MOVL C09799 V=800.0 PL=0
MOVL C09800 V=800.0 PL=0
MOVL C09801 V=800.0 PL=0
MOVL C09802 V=800.0 PL=0
MOVL C09803 V=800.0 PL=0
MOVL C09804 V=800.0 PL=0
MOVL C09805 V=800.0 PL=0
MOVL C09806 V=800.0 PL=0
MOVL C09807 V=800.0 PL=0
MOVL C09808 V=800.0 PL=0
MOVL C09809 V=800.0 PL=0
MOVL C09810 V=800.0 PL=0
MOVL C09811 V=800.0 PL=0
MOVL C09812 V=800.0 PL=0
MOVL C09813 V=800.0 PL=0
MOVL C09814 V=800.0 PL=0
MOVL C09815 V=800.0 PL=0
MOVL C09816 V=800.0 PL=0
MOVL C09817 V=800.0 PL=0
MOVL C09818 V=800.0 PL=0
MOVL C09819 V=800.0 PL=0
MOVL C09820 V=800.0 PL=0
MOVL C09821 V=800.0 PL=0
MOVL C09822 V=800.0 PL=0
MOVL C09823 V=800.0 PL=0
MOVL C09824 V=800.0 PL=0
MOVL C09825 V=800.0 PL=0
MOVL C09826 V=800.0 PL=0
MOVL C09827 V=800.0 PL=0
MOVL C09828 V=800.0 PL=0
MOVL C09829 V=800.0 PL=0
MOVL C09830 V=800.0 PL=0
MOVL C09831 V=800.0 PL=0
MOVL C09832 V=800.0 PL=0
MOVL C09833 V=800.0 PL=0
MOVL C09834 V=800.0 PL=0
MOVL C09835 V=800.0 PL=0
MOVL C09836 V=800.0 PL=0
MOVL C09837 V=800.0 PL=0
MOVL C09838 V=800.0 PL=0
MOVL C09839 V=800.0 PL=0
MOVL C09840 V=800.0 PL=0
MOVL C09841 V=800.0 PL=0
MOVL C09842 V=800.0 PL=0
MOVL C09843 V=800.0 PL=0
MOVL C09844 V=800.0 PL=0
MOVL C09845 V=800.0 PL=0
MOVL C09846 V=800.0 PL=0
MOVL C09847 V=800.0 PL=0
MOVL C09848 V=800.0 PL=0
MOVL C09849 V=800.0 PL=0
MOVL C09850 V=800.0 PL=0
MOVL C09851 V=800.0 PL=0
MOVL C09852 V=800.0 PL=0
MOVL C09853 V=800.0 PL=0
MOVL C09854 V=800.0 PL=0
MOVL C09855 V=800.0 PL=0
MOVL C09856 V=800.0 PL=0
MOVL C09857 V=800.0 PL=0
MOVL C09858 V=800.0 PL=0
MOVL C09859 V=800.0 PL=0
MOVL C09860 V=800.0 PL=0
MOVL C09861 V=800.0 PL=0
MOVL C09862 V=800.0 PL=0
MOVL C09863 V=800.0 PL=0
MOVL C09864 V=800.0 PL=0
MOVL C09865 V=800.0 PL=0
MOVL C09866 V=800.0 PL=0
MOVL C09867 V=800.0 PL=0
MOVL C09868 V=800.0 PL=0
MOVL C09869 V=800.0 PL=0
MOVL C09870 V=800.0 PL=0
MOVL C09871 V=800.0 PL=0
MOVL C09872 V=800.0 PL=0
MOVL C09873 V=800.0 PL=0
MOVL C09874 V=800.0 PL=0
MOVL C09875 V=800.0 PL=0
MOVL C09876 V=800.0 PL=0
MOVL C09877 V=800.0 PL=0
MOVL C09878 V=800.0 PL=0
MOVL C09879 V=800.0 PL=0
MOVL C09880 V=800.0 PL=0
MOVL C09881 V=800.0 PL=0
MOVL C09882 V=800.0 PL=0
MOVL C09883 V=800.0 PL=0
MOVL C09884 V=800.0 PL=0
MOVL C09885 V=800.0 PL=0
MOVL C09886 V=800.0 PL=0
MOVL C09887 V=800.0 PL=0
MOVL C09888 V=800.0 PL=0
MOVL C09889 V=800.0 PL=0
MOVL C09890 V=800.0 PL=0
MOVL C09891 V=800.0 PL=0
MOVL C09892 V=800.0 PL=0
MOVL C09893 V=800.0 PL=0
MOVL C09894 V=800.0 PL=0
MOVL C09895 V=800.0 PL=0
MOVL C09896 V=800.0 PL=0
MOVL C09897 V=800.0 PL=0
MOVL C09898 V=800.0 PL=0
MOVL C09899 V=800.0 PL=0
MOVL C09900 V=800.0 PL=0
MOVL C09901 V=800.0 PL=0
MOVL C09902 V=800.0 PL=0
MOVL C09903 V=800.0 PL=0
MOVL C09904 V=800.0 PL=0
MOVL C09905 V=800.0 PL=0
MOVL C09906 V=800.0 PL=0
MOVL C09907 V=800.0 PL=0
MOVL C09908 V=800.0 PL=0
MOVL C09909 V=800.0 PL=0
MOVL C09910 V=800.0 PL=0
MOVL C09911 V=800.0 PL=0
MOVL C09912 V=800.0 PL=0
MOVL C09913 V=800.0 PL=0
MOVL C09914 V=800.0 PL=0
MOVL C09915 V=800.0 PL=0
MOVL C09916 V=800.0 PL=0
MOVL C09917 V=800.0 PL=0
MOVL C09918 V=800.0 PL=0
MOVL C09919 V=800.0 PL=0
MOVL C09920 V=800.0 PL=0
MOVL C09921 V=800.0 PL=0
MOVL C09922 V=800.0 PL=0
MOVL C09923 V=800.0 PL=0
MOVL C09924 V=800.0 PL=0
MOVL C09925 V=800.0 PL=0
MOVL C09926 V=800.0 PL=0
MOVL C09927 V=800.0 PL=0
MOVL C09928 V=800.0 PL=0
MOVL C09929 V=800.0 PL=0
MOVL C09930 V=800.0 PL=0
MOVL C09931 V=800.0 PL=0
MOVL C09932 V=800.0 PL=0
MOVL C09933 V=800.0 PL=0
MOVL C09934 V=800.0 PL=0
MOVL C09935 V=800.0 PL=0
MOVL C09936 V=800.0 PL=0
MOVL C09937 V=800.0 PL=0
MOVL C09938 V=800.0 PL=0
MOVL C09939 V=800.0 PL=0
MOVL C09940 V=800.0 PL=0
MOVL C09941 V=800.0 PL=0
MOVL C09942 V=800.0 PL=0
MOVL C09943 V=800.0 PL=0
MOVL C09944 V=800.0 PL=0
MOVL C09945 V=800.0 PL=0
MOVL C09946 V=800.0 PL=0
MOVL C09947 V=800.0 PL=0
MOVL C09948 V=800.0 PL=0
MOVL C09949 V=800.0 PL=0
MOVL C09950 V=800.0 PL=0
MOVL C09951 V=800.0 PL=0
MOVL C09952 V=800.0 PL=0
MOVL C09953 V=800.0 PL=0
MOVL C09954 V=800.0 PL=0
MOVL C09955 V=800.0 PL=0
MOVL C09956 V=800.0 PL=0
MOVL C09957 V=800.0 PL=0
MOVL C09958 V=800.0 PL=0
MOVL C09959 V=800.0 PL=0
MOVL C09960 V=800.0 PL=0
MOVL C09961 V=800.0 PL=0
MOVL C09962 V=800.0 PL=0
MOVL C09963 V=800.0 PL=0
MOVL C09964 V=800.0 PL=0
MOVL C09965 V=800.0 PL=0
MOVL C09966 V=800.0 PL=0
MOVL C09967 V=800.0 PL=0
MOVL C09968 V=800.0 PL=0
MOVL C09969 V=800.0 PL=0
MOVL C09970 V=800.0 PL=0
MOVL C09971 V=800.0 PL=0
MOVL C09972 V=800.0 PL=0
MOVL C09973 V=800.0 PL=0
MOVL C09974 V=800.0 PL=0
MOVL C09975 V=800.0 PL=0
MOVL C09976 V=800.0 PL=0
MOVL C09977 V=800.0 PL=0
MOVL C09978 V=800.0 PL=0
MOVL C09979 V=800.0 PL=0
MOVL C09980 V=800.0 PL=0
MOVL C09981 V=800.0 PL=0
MOVL C09982 V=800.0 PL=0
MOVL C09983 V=800.0 PL=0
MOVL C09984 V=800.0 PL=0
MOVL C09985 V=800.0 PL=0
MOVL C09986 V=800.0 PL=0
MOVL C09987 V=800.0 PL=0
MOVL C09988 V=800.0 PL=0
MOVL C09989 V=800.0 PL=0
MOVL C09990 V=800.0 PL=0
MOVL C09991 V=800.0 PL=0
MOVL C09992 V=800.0 PL=0
MOVL C09993 V=800.0 PL=0
MOVL C09994 V=800.0 PL=0
MOVL C09995 V=800.0 PL=0
MOVL C09996 V=800.0 PL=0
CALL JOB:A_ROOF_SIDE_0617_2_PAINT_45
END
